// LS Electric XG5000 project: SmartSorter
// PLC LSPLC

PROGRAM NewProgram (task: 스캔 프로그램)

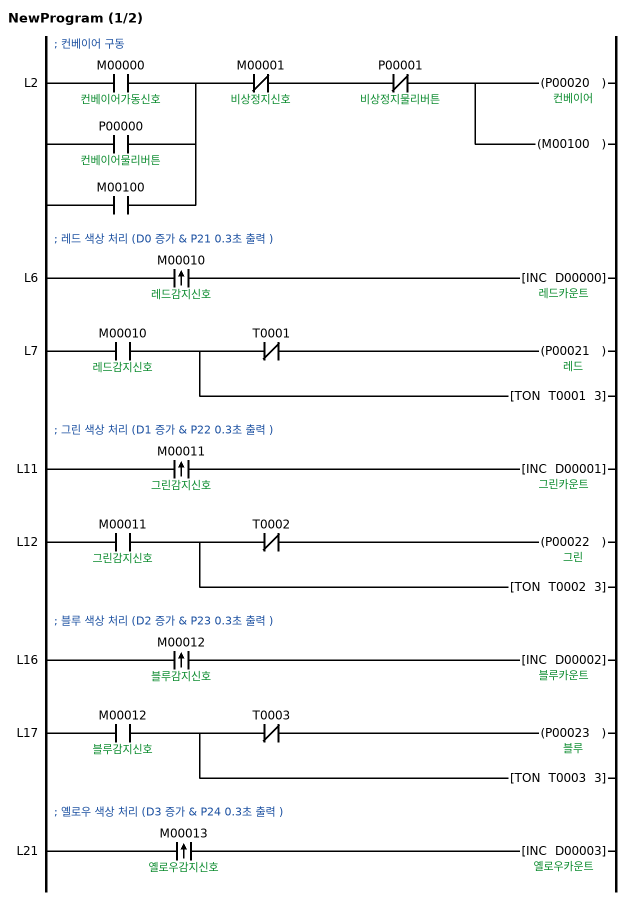
// 컨베이어 구동
; L2
LOAD      M00000	// 컨베이어가동신호
OR        P00000	// 컨베이어물리버튼
OR        M00100
AND NOT   M00001	// 비상정지신호
AND NOT   P00001	// 비상정지물리버튼
OUT       P00020	// 컨베이어
OUT       M00100
// 레드 색상 처리 (D0 증가 & P21 0.3초 출력 )
; L6
LOADP     M00010	// 레드감지신호
INC       D00000	// 레드카운트
; L7
LOAD      M00010	// 레드감지신호
MPUSH
AND NOT   T0001
OUT       P00021	// 레드
MPOP
TON       T0001 3
// 그린 색상 처리 (D1 증가 & P22 0.3초 출력 )
; L11
LOADP     M00011	// 그린감지신호
INC       D00001	// 그린카운트
; L12
LOAD      M00011	// 그린감지신호
MPUSH
AND NOT   T0002
OUT       P00022	// 그린
MPOP
TON       T0002 3
// 블루 색상 처리 (D2 증가 & P23 0.3초 출력 )
; L16
LOADP     M00012	// 블루감지신호
INC       D00002	// 블루카운트
; L17
LOAD      M00012	// 블루감지신호
MPUSH
AND NOT   T0003
OUT       P00023	// 블루
MPOP
TON       T0003 3
// 옐로우 색상 처리 (D3 증가 & P24 0.3초 출력 )
; L21
LOADP     M00013	// 옐로우감지신호
INC       D00003	// 옐로우카운트

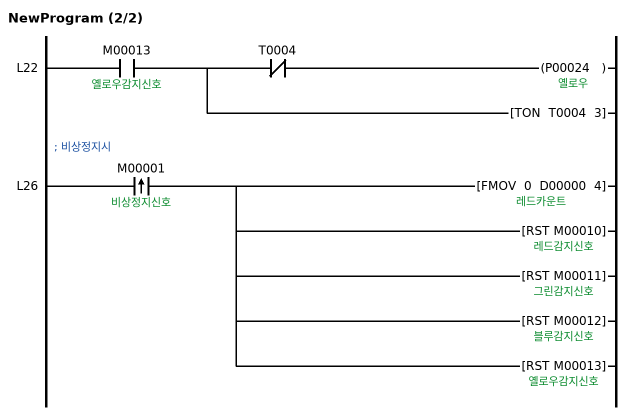
; L22
LOAD      M00013	// 옐로우감지신호
MPUSH
AND NOT   T0004
OUT       P00024	// 옐로우
MPOP
TON       T0004 3
// 비상정지시
; L26
LOADP     M00001	// 비상정지신호
FMOV      0 D00000 4	// 레드카운트
RST       M00010	// 레드감지신호
RST       M00011	// 그린감지신호
RST       M00012	// 블루감지신호
RST       M00013	// 옐로우감지신호